{attribute 'qualified_only'}
{attribute 'strict'}
TYPE ProfileLimitsEnum :
(
	acc0_acc1_vel,
  vel, 
  acc0,
  acc1,
  acc0_acc1,
  acc0_vel,
  acc1_vel,
  none
);
END_TYPE

(* stored: Version 1.1.0.1, ProductVersion 3.1.4024.6
   DUT ProfileLimitsEnum: Id {bd5b0c3f-6bf6-4746-af09-80103c0606f6} *)
